Staubli VAL3: PublicProg.dtx

public mdesc mNomSpeed
public string sfliePath
string sContent
